// TIA Portal V16 export
// export: Created 2022-02-28T20:45:44.916034Z, ExportSetting WithDefaults, DisplayName Totally Integrated Automation Portal, DisplayVersion V16, DisplayName TIA Portal Version Control Interface, DisplayVersion V16, DisplayName TIA Portal Openness, DisplayVersion V16, DisplayName STEP 7 Professional, DisplayVersion V16, DisplayName STEP 7 Safety, DisplayVersion V16, DisplayName WinCC Advanced, DisplayVersion V16
FUNCTION "04_Control_Codigos1" : Void   // FC4, LAD
{ S7_Optimized_Access := 'TRUE' }
VERSION : 0.1
// stored: AutoNumber true, IsIECCheckEnabled false, SetENOAutomatically false, UDAEnableTagReadback false
   VAR_IN_OUT
      Registro : "UDT_DatosProd";
   END_VAR
   VAR_TEMP
      i : Int;
      DNC : Bool;
   END_VAR
   VAR_TEMP   // added for the SCL form of the ladder/FBD networks
      _w1 : Bool;
   END_VAR
BEGIN

REGION Network 1
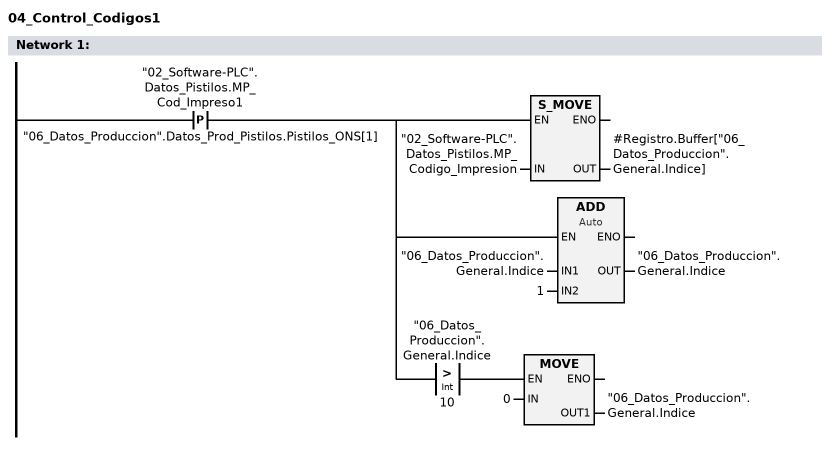
   RUNG wire#powerrail
      P_Contact(operand := "02_Software-PLC".Datos_Pistilos.MP_Cod_Impreso1, bit := "06_Datos_Produccion".Datos_Prod_Pistilos.Pistilos_ONS[1])
      wire#w1
      S_Move(in := "02_Software-PLC".Datos_Pistilos.MP_Codigo_Impresion, out => #Registro.Buffer["06_Datos_Produccion".General.Indice])
   END_RUNG
   RUNG wire#w1
      Add(in1 := "06_Datos_Produccion".General.Indice, in2 := 1, out => "06_Datos_Produccion".General.Indice)
   END_RUNG
   RUNG wire#w1
      { S7_Templates := "SrcType := Int" } GT_Contact(in1 := "06_Datos_Produccion".General.Indice, in2 := 10)
      Move(in := 0, out1 => "06_Datos_Produccion".General.Indice)
   END_RUNG
   // the same network as SCL:
   #_w1 := "02_Software-PLC".Datos_Pistilos.MP_Cod_Impreso1 AND NOT "06_Datos_Produccion".Datos_Prod_Pistilos.Pistilos_ONS[1];   // rising edge of "02_Software-PLC".Datos_Pistilos.MP_Cod_Impreso1
   "06_Datos_Produccion".Datos_Prod_Pistilos.Pistilos_ONS[1] := "02_Software-PLC".Datos_Pistilos.MP_Cod_Impreso1;
   IF #_w1 THEN
       #Registro.Buffer["06_Datos_Produccion".General.Indice] := "02_Software-PLC".Datos_Pistilos.MP_Codigo_Impresion;
       "06_Datos_Produccion".General.Indice := "06_Datos_Produccion".General.Indice + 1;
   END_IF;
   IF #_w1 AND ("06_Datos_Produccion".General.Indice > 10) THEN
       "06_Datos_Produccion".General.Indice := 0;
   END_IF;
END_REGION

REGION Network 3 (SCL)
   IF #Registro.Entradas.Extraccion THEN 
       #Registro.Salidas.Ext_Dn := 1;

       FOR #i := 0 TO #Registro.Entradas.Longitud DO

           IF #Registro.Buffer[#i] = #Registro.valor_Camara THEN

               #Registro.Buffer[#i] := '';
           ELSE
               #DNC := 1;

               EXIT;
           END_IF;

       END_FOR;

   END_IF;
END_REGION
END_FUNCTION
